INTERFACE ITF_ControlE_TE1_HMI_Connector EXTENDS ITF_BaseControlElement_HMI_Connector

END_INTERFACE

(* stored: Version 1.1.0.1, ProductVersion 3.1.4024.15
   Itf ITF_ControlE_TE1_HMI_Connector: Id {5196c1fa-c67c-4f77-a6a5-461451ac3161} *)
